Universal Robots PolyScope program: Step Corner Right Down Around under.urp

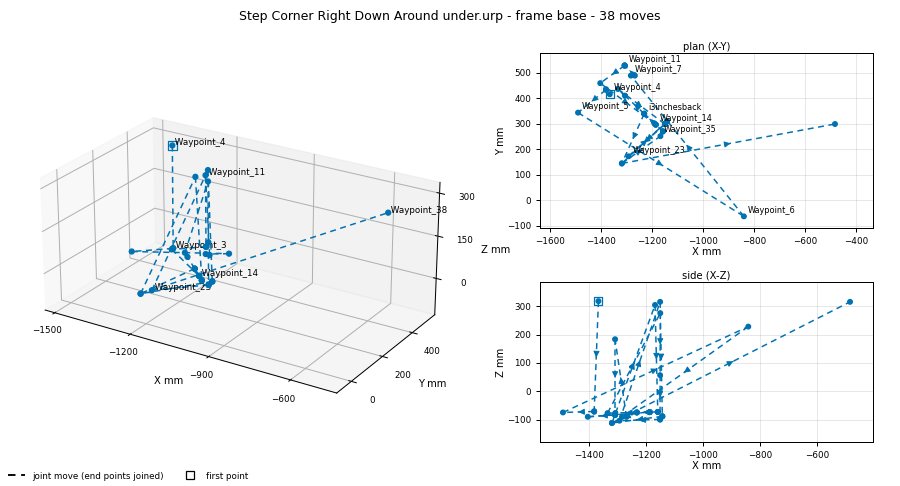
[picture p0: tool path of Step Corner Right Down Around under.urp in frame base, 38 of 38 moves have a stored position in this frame; points joined in program order, loops and branches not executed]
Program Step Corner Right Down Around under (installation=default directory=/programs createdIn=5.21.3 lastSavedIn=5.21.3 robotSerialNumber=20246801938)
Calibrated DH parameters: a=[-0.000071, -0.790281, -0.600694, 0.000061, -0.000039, 0]; d=[0.236272, 604.465945, 132.116513, -736.382239, 0.159268, 0.154005]; alpha=[1.570254, -0.000567, 0.000559, 1.571709, -1.56999, 0]; deltaTheta=[0, -0.409357, 7.293326, -0.600784, -0.000001, -0.000001]
InitVariablesNode
Robot Program (runOnlyOnce=false)
  Folder dummy points
    MoveJ speed 60 deg/s, acceleration 80 deg/s^2 (useActiveTCP=true optimoveEnabled=false optiMoveSpeed=0.3 optiMoveAcceleration=0.09) feature=Base
      'wrist from the bottom'
      Waypoint Waypoint_4: TCP in base x=-1367.411 y=416.277 z=317.19 mm, rx=-0.7822 ry=-1.6629 rz=1.6144 rad; joints [-34.032, -39.596, 100.247, 115.549, -109.961, -91.263] deg; TCP offset x=-9.5 y=-328 z=105.73 mm, rx=1.2092 ry=-1.2092 rz=1.2092 rad
      Waypoint Waypoint_3: TCP in base x=-1382.402 y=435.382 z=-70.39 mm, rx=-0.7822 ry=-1.6629 rz=1.6144 rad; joints [-34.456, -15.059, 88.261, 103.003, -109.526, -91.251] deg
      Waypoint Waypoint_2: TCP in base x=-1382.402 y=435.382 z=-70.39 mm, rx=-0.4004 ry=-0.9435 rz=2.0176 rad; joints [-30.86, 0.221, 70.994, 104.887, -113.107, -49.94] deg
      Waypoint Waypoint_1: TCP in base x=-1382.402 y=433.691 z=-70.39 mm, rx=0.0561 ry=-0.0602 rz=2.256 rad; joints [-21.342, 13.524, 42.978, 119.463, -119.274, -3.474] deg
      Waypoint Waypoint_5: TCP in base x=-1491.969 y=344.099 z=-73.835 mm, rx=0.0561 ry=-0.0602 rz=2.256 rad; joints [-15.949, 21.497, 21.478, 132.739, -124.647, -3.926] deg
    MoveJ speed 60 deg/s, acceleration 80 deg/s^2 (useActiveTCP=true optimoveEnabled=false optiMoveSpeed=0.3 optiMoveAcceleration=0.09) feature=Base
      'align for legback'
      Waypoint Waypoint_6: TCP in base x=-841.02 y=-62.951 z=227.762 mm, rx=0.0004 ry=-0.0577 rz=0.6541 rad; joints [-156.731, -147.195, -97.361, -118.678, 75.795, 179.795] deg
      Waypoint Waypoint_7: TCP in base x=-1284.619 y=489.384 z=-89.321 mm, rx=0.0004 ry=-0.0577 rz=0.6541 rad; joints [-185.005, -195.006, -8.043, -161.208, 47.526, 181.864] deg
      Waypoint Waypoint_8: TCP in base x=-1268.871 y=489.382 z=-89.349 mm, rx=-0.0027 ry=-0.0573 rz=0.5465 rad; joints [-185.786, -198.817, 0.384, -165.501, 52.897, 181.363] deg
      'this is the farthest it can go on the right'
    MoveJ speed 60 deg/s, acceleration 80 deg/s^2 (useActiveTCP=true optimoveEnabled=false optiMoveSpeed=0.3 optiMoveAcceleration=0.09) feature=Base
      'wrist from the bottom'
      Waypoint Waypoint_11: TCP in base x=-1308.945 y=528.973 z=183.362 mm, rx=-0.7814 ry=-1.6613 rz=1.6156 rad; joints [-41.138, -31.537, 98.613, 109.272, -102.866, -90.693] deg
      Waypoint Waypoint_10: TCP in base x=-1308.945 y=528.973 z=-82.602 mm, rx=-0.7788 ry=-1.6566 rz=1.6193 rad; joints [-41.15, -14.573, 89.924, 100.994, -102.846, -90.409] deg
      Waypoint Waypoint_9: TCP in base x=-1308.945 y=528.973 z=-82.602 mm, rx=-0.2844 ry=-0.7211 rz=2.0918 rad; joints [-34.731, 4.177, 67.194, 104.837, -109.247, -37.582] deg
      Waypoint Waypoint_12: TCP in base x=-1308.945 y=528.973 z=-82.602 mm, rx=0.0382 ry=-0.095 rz=2.1962 rad; joints [-26.714, 12.257, 48.872, 114.831, -117.243, -5.085] deg
      Waypoint Waypoint_13: TCP in base x=-1404.769 y=459.807 z=-89.048 mm, rx=0.0382 ry=-0.095 rz=2.1962 rad; joints [-21.899, 16.949, 35.307, 123.498, -122.043, -5.48] deg
    MoveJ speed 60 deg/s, acceleration 80 deg/s^2 (useActiveTCP=true optimoveEnabled=false optiMoveSpeed=0.3 optiMoveAcceleration=0.09) feature=Base
      'align legback at 41 inches from corner'
      Waypoint Waypoint_14: TCP in base x=-1186.908 y=296.959 z=-72.677 mm, rx=0.0004 ry=-0.0577 rz=0.6541 rad; joints [-177.362, -178.188, -47.228, -138.41, 55.173, 181.179] deg
      Waypoint Waypoint_15: TCP in base x=-1186.908 y=296.959 z=-72.677 mm, rx=0.0051 ry=-0.0581 rz=0.8157 rad; joints [-176.136, -176.438, -52.018, -135.832, 47.157, 181.909] deg
      Waypoint i3inchesback: TCP in base x=-1232.315 y=339.713 z=-73.791 mm, rx=0.0051 ry=-0.0581 rz=0.8157 rad; joints [-178.036, -179.66, -43.462, -141.304, 45.258, 182.108] deg
      Waypoint i7inchesback: TCP in base x=-1307.925 y=410.908 z=-75.645 mm, rx=0.0051 ry=-0.0581 rz=0.8157 rad; joints [-180.924, -188.186, -22.525, -153.953, 42.367, 182.436] deg
      Waypoint asfaraswecango: TCP in base x=-1335.405 y=436.787 z=-76.32 mm, rx=0.0051 ry=-0.0581 rz=0.8157 rad; joints [-181.892, -198.249, 0.21, -166.712, 41.391, 182.553] deg
      '8 inches back is as far as it can go'
      'good clearance on the wrist not hitting'
    MoveJ speed 60 deg/s, acceleration 80 deg/s^2 (useActiveTCP=true optimoveEnabled=false optiMoveSpeed=0.3 optiMoveAcceleration=0.09) feature=Base
      '41 inches away right down and around  (normal)'
      SuppressedNode
        Waypoint Waypoint_16: TCP in base x=-1152.776 y=298.966 z=176.739 mm, rx=-0.7814 ry=-1.6613 rz=1.6156 rad; joints [-35.748, -35.335, 119.924, 91.649, -108.243, -91.062] deg
      Waypoint Waypoint_19: TCP in base x=-1150.141 y=298.643 z=275.063 mm, rx=-0.7684 ry=-1.7225 rz=1.7195 rad; joints [-38.296, -44.064, 121.651, 102.229, -100.056, -90.146] deg
      Waypoint Waypoint_18: TCP in base x=-1150.657 y=299.267 z=57.141 mm, rx=-0.7684 ry=-1.7225 rz=1.7195 rad; joints [-38.317, -27.522, 116.556, 90.779, -100.028, -90.16] deg
      Waypoint Waypoint_20: TCP in base x=-1151.009 y=299.695 z=-98.245 mm, rx=-0.7684 ry=-1.7225 rz=1.7195 rad; joints [-38.333, -16.247, 110.211, 85.848, -100.006, -90.167] deg
      Waypoint Waypoint_21: TCP in base x=-1151.009 y=299.695 z=-98.245 mm, rx=-0.4308 ry=-0.9713 rz=2.1266 rad; joints [-33.127, -1.565, 95.44, 85.92, -105.204, -49.184] deg
      Waypoint Waypoint_22: TCP in base x=-1151.009 y=299.695 z=-98.245 mm, rx=-0.0079 ry=-0.0286 rz=2.2985 rad; joints [-18.881, 6.735, 75.564, 97.447, -119.451, -1.573] deg
      Waypoint Waypoint_23: TCP in base x=-1293.478 y=172.756 z=-102.692 mm, rx=-0.0079 ry=-0.0286 rz=2.2985 rad; joints [-9.985, 9.351, 61.312, 109.038, -128.348, -1.618] deg
      SuppressedNode
        Waypoint Waypoint_17: TCP in base x=-1153 y=301.142 z=-78.491 mm, rx=-0.6898 ry=-1.7732 rz=1.761 rad; joints [-40.029, -17.338, 109.154, 86.957, -93.795, -90.095] deg
    MoveJ speed 60 deg/s, acceleration 80 deg/s^2 (useActiveTCP=true optimoveEnabled=false optiMoveSpeed=0.3 optiMoveAcceleration=0.09) feature=Base
      'try the right down and around while already elbow shoulder flipped. save time in between weld segments.'
      SuppressedNode
        Waypoint Waypoint_24: TCP in base x=-1159.383 y=294.639 z=314.427 mm, rx=-0.763 ry=-1.7686 rz=1.7098 rad; joints [-189.584, -110.898, -118.053, -130.576, -52.569, 87.903] deg
      Waypoint Waypoint_25: TCP in base x=-1150.667 y=299.412 z=314.716 mm, rx=-0.763 ry=-1.7686 rz=1.7098 rad; joints [-190.036, -110.575, -118.548, -130.408, -53.021, 87.908] deg
      Waypoint Waypoint_26: TCP in base x=-1142.969 y=309.681 z=-87.506 mm, rx=-0.763 ry=-1.7686 rz=1.7098 rad; joints [-190.869, -138.561, -121.1, -99.861, -53.852, 87.895] deg
      Waypoint Waypoint_27: TCP in base x=-1142.969 y=309.681 z=-87.506 mm, rx=-0.3723 ry=-0.8733 rz=2.1834 rad; joints [-185.608, -157.456, -110.732, -91.291, -48.6, 136.169] deg
      Waypoint Waypoint_28: TCP in base x=-1142.969 y=309.681 z=-87.506 mm, rx=-0.042 ry=-0.1145 rz=2.3191 rad; joints [-176.856, -164.495, -97.958, -96.936, -39.853, 173.997] deg
      Waypoint Waypoint_29: TCP in base x=-1319.931 y=144.753 z=-110.859 mm, rx=-0.042 ry=-0.1145 rz=2.3191 rad; joints [-168.827, -168.671, -81.313, -109.278, -31.832, 173.844] deg
    MoveJ speed 60 deg/s, acceleration 80 deg/s^2 (useActiveTCP=true optimoveEnabled=false optiMoveSpeed=0.3 optiMoveAcceleration=0.09) feature=Base
      'left side down and around'
      Waypoint Waypoint_35: TCP in base x=-1168.534 y=251.879 z=303.712 mm, rx=-1.4388 ry=-0.6695 rz=0.6003 rad; joints [-161.388, -128.913, -89.606, -145.038, 61.894, 92.57] deg
      Waypoint Waypoint_34: TCP in base x=-1158.879 y=270.56 z=-71.906 mm, rx=-1.4388 ry=-0.6695 rz=0.6003 rad; joints [-162.149, -147.253, -91.84, -124.494, 61.136, 92.631] deg
      Waypoint Waypoint_33: TCP in base x=-1158.879 y=270.56 z=-71.906 mm, rx=-0.7017 ry=-0.3606 rz=0.7543 rad; joints [-166.587, -162.657, -80.402, -120.702, 56.7, 138.104] deg
      Waypoint Waypoint_32: TCP in base x=-1158.879 y=270.56 z=-71.906 mm, rx=0.0031 ry=-0.059 rz=0.8157 rad; joints [-174.873, -174.753, -56.691, -132.759, 48.42, 181.66] deg
      Waypoint Waypoint_30: TCP in base x=-1186.908 y=296.959 z=-72.677 mm, rx=0.0051 ry=-0.0581 rz=0.8157 rad; joints [-176.136, -176.438, -52.018, -135.832, 47.157, 181.909] deg
      Waypoint Waypoint_31: TCP in base x=-1232.315 y=339.713 z=-73.791 mm, rx=0.0051 ry=-0.0581 rz=0.8157 rad; joints [-178.036, -179.66, -43.462, -141.304, 45.258, 182.108] deg
    MoveJ speed 60 deg/s, acceleration 80 deg/s^2 (useActiveTCP=true optimoveEnabled=false optiMoveSpeed=0.3 optiMoveAcceleration=0.09) feature=Base
      'ramping endpoints'
      Waypoint Waypoint_36: TCP in base x=-1232.315 y=339.713 z=-73.791 mm, rx=-0.1375 ry=-0.1153 rz=0.8103 rad; joints [-176.519, -176.703, -50.605, -136.703, 46.753, 173.18] deg
      'above is ramping for backaway on theright side of box'
      Waypoint Waypoint_37: TCP in base x=-1319.931 y=144.753 z=-110.859 mm, rx=-0.1205 ry=-0.295 rz=2.3058 rad; joints [-170.257, -167.221, -85.468, -106.599, -33.26, 164.949] deg
      'above is ramping for the backaway on left side of box'
    MoveJ speed 60 deg/s, acceleration 80 deg/s^2 (useActiveTCP=true optimoveEnabled=false optiMoveSpeed=0.3 optiMoveAcceleration=0.09) feature=Base
      'approach points'
      Waypoint Waypoint_38: TCP in base x=-483.576 y=299.412 z=314.716 mm, rx=-0.763 ry=-1.7686 rz=1.7098 rad; joints [-222.644, -81.791, -155.216, -122.625, -85.615, 88.172] deg; TCP offset x=4.51 y=-328 z=105.73 mm, rx=1.2092 ry=-1.2092 rz=1.2092 rad
      'above is approach point for right weld'
